(* PLC project SafeLOGIC-1, BrAutomation SafeDESIGNER  4.2.2.18 *)
(* stored: companyURL http://www.br-automation.com, creationDateTime Wed Apr 05 12:57:43 2017 *)

PROGRAM Main

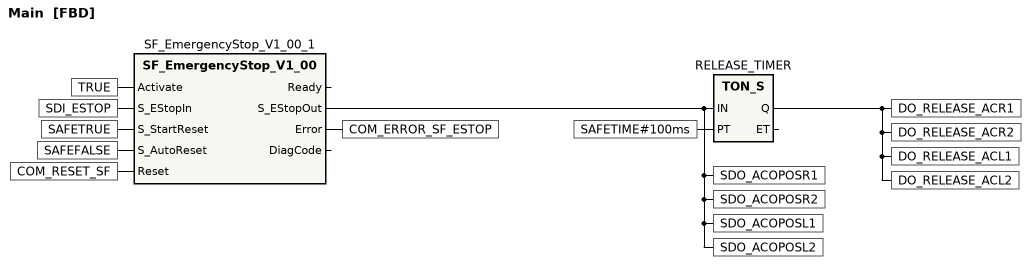
(* FBD diagram, written out as Structured Text *)
SF_EmergencyStop_V1_00_1(Activate := TRUE, S_EStopIn := SDI_ESTOP, S_StartReset := SAFETRUE, S_AutoReset := SAFEFALSE, Reset := COM_RESET_SF);
COM_ERROR_SF_ESTOP := SF_EmergencyStop_V1_00_1.Error;
SDO_ACOPOSR1 := SF_EmergencyStop_V1_00_1.S_EStopOut;
SDO_ACOPOSR2 := SF_EmergencyStop_V1_00_1.S_EStopOut;
SDO_ACOPOSL1 := SF_EmergencyStop_V1_00_1.S_EStopOut;
RELEASE_TIMER(IN := SF_EmergencyStop_V1_00_1.S_EStopOut, PT := SAFETIME#100ms);
DO_RELEASE_ACR1 := RELEASE_TIMER.Q;
SDO_ACOPOSL2 := SF_EmergencyStop_V1_00_1.S_EStopOut;
DO_RELEASE_ACR2 := RELEASE_TIMER.Q;
DO_RELEASE_ACL1 := RELEASE_TIMER.Q;
DO_RELEASE_ACL2 := RELEASE_TIMER.Q;
END_PROGRAM
